(* IEC 61131-3 sources: axopen.templates/axopen.template.simple/ax/templates-sources/unit/Data/_managers_, 3 files *)

(* ---- ProcessDataManger.st ---- *)
NAMESPACE axosimple.UnitTemplate
    USING axosimple;
    USING AXOpen.Data;
    USING AXOpen.Core;
    USING System.Strings;

    {S7.extern=ReadWrite}
    CLASS ProcessDataManager
        EXTENDS AXOpen.Data.AxoDataFragmentExchange
        VAR PUBLIC
            {#ix-attr:[AXOpen.Data.AxoDataFragmentAttribute]}
            Shared : axosimple.SharedDataExchange;
            {#ix-attr:[AXOpen.Data.AxoDataFragmentAttribute]}
            Data : ProcessDataExchange;
        END_VAR

        METHOD PUBLIC OVERRIDE Run
            VAR_INPUT
                parent : IAxoObject;
            END_VAR
              Shared.Run(THIS);
              Data.Run(THIS);
              SUPER.Run(parent := parent);
        END_METHOD
    END_CLASS
END_NAMESPACE

(* ---- TechnologyDataExchange.st ---- *)
NAMESPACE axosimple.UnitTemplate
    USING axosimple;
    USING AXOpen.Data;
    USING AXOpen.Core;
    USING System.Strings;

    {S7.extern=ReadWrite}
    CLASS TechnologyDataExchange
        EXTENDS AXOpen.Data.AxoDataExchange
        VAR PUBLIC
            {#ix-generic:TOnline}
            {#ix-generic:TPlain as POCO}
            {#ix-attr:[AXOpen.Data.AxoDataEntityAttribute]}
            {#ix-attr:[Container(Layout.Stack)]}
            {#ix-set:AttributeName = "<#UnitTemplate#>"}
            Payload : TechnologyDataPayload;
        END_VAR
    END_CLASS
END_NAMESPACE

(* ---- TechnologyDataManager.st ---- *)
NAMESPACE axosimple.UnitTemplate
    USING axosimple;
    USING AXOpen.Data;
    USING AXOpen.Core;
    USING System.Strings;

    {S7.extern=ReadWrite}
    CLASS TechnologyDataManager
        EXTENDS AXOpen.Data.AxoDataFragmentExchange
        VAR PUBLIC
            {#ix-attr:[AXOpen.Data.AxoDataFragmentAttribute]}
            Shared : axosimple.TechnologySharedDataExchange;
            {#ix-attr:[AXOpen.Data.AxoDataFragmentAttribute]}
            Data : TechnologyDataExchange;
        END_VAR

        METHOD PUBLIC OVERRIDE Run
            VAR_INPUT
                parent : IAxoObject;
            END_VAR
              Shared.Run(THIS);
              Data.Run(THIS);
              SUPER.Run(parent := parent);
        END_METHOD
    END_CLASS
END_NAMESPACE
